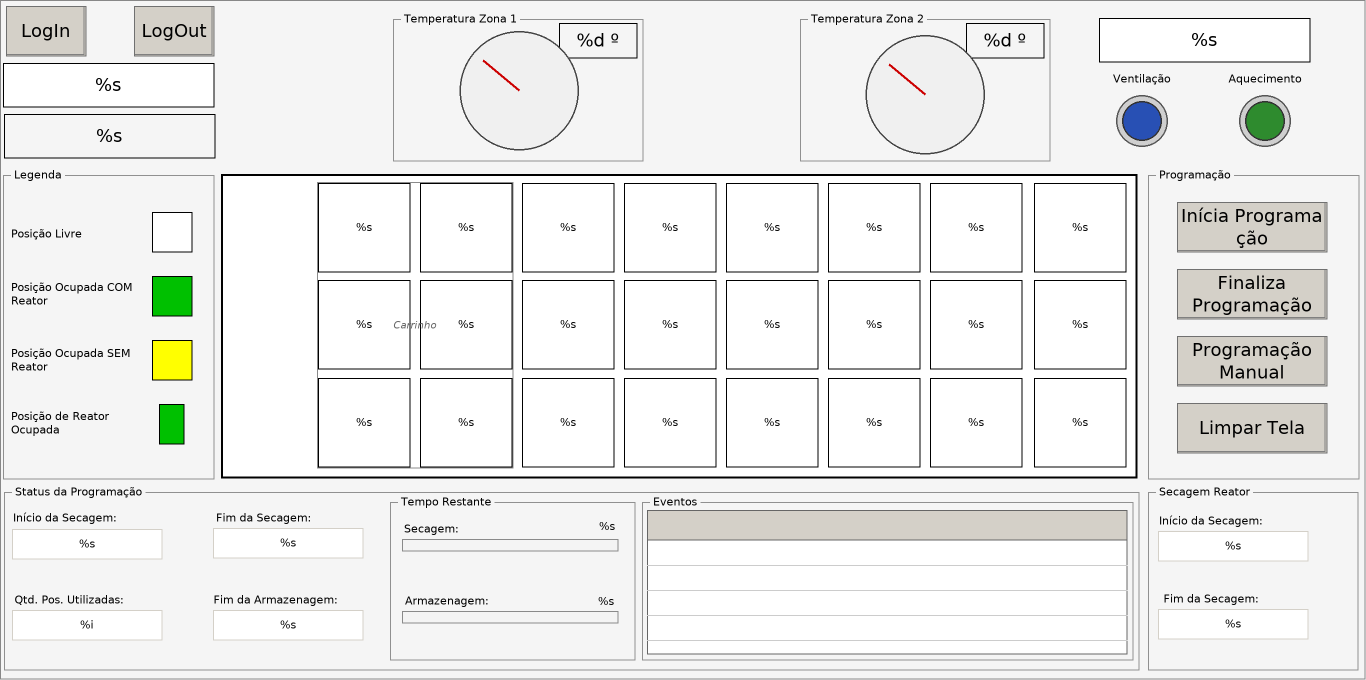
VISUALIZATION Estufa1  // 1366x680
    GroupBox (1148,484 210x186), "Secagem Reator", invisible if: GVL_P.bCarrinhoReator1
        Label (10,100 106x30), "Fim da Secagem:"
        Textfield (10,125 150x30), "%s", text variable: GVL_P.arrStatusEstufas[0].statusFimSecagem
    GroupBox (3,167 211x312), "Legenda"
        RoundedRectangle (149,173 40x40)
        RoundedRectangle (149,45 40x40)
        RoundedRectangle (156,237 25x40)
    GroupBox (800,11 250x150), "Temperatura Zona 2"
        Rectangle (166,12 78x35), "%d º", text variable: GVL.zona2atual_019
    GroupBox (393,11 250x150), "Temperatura Zona 1"
        Rectangle (166,12 78x35), "%d º", text variable: GVL.zona1atual_019
    GroupBox (4,484 1135x186), "Status da Programação"
        Label (209,19 101x30), "Fim da Secagem:"
        Label (209,101 125x30), "Fim da Armazenagem:"
        Label (8,101 114x30), "Qtd. Pos. Utilizadas:"
        GroupBox (638,10 491x166), "Eventos"
            Table (5,16 480x144), data array: GVL_P.arrLogEstufa19
                p3854506369: GVL_P.arrLogEstufa19[INDEX]
            InvisibleInput (6,17 431x142)
                OnMouseClick: OpenDialog Dialog=addComment, OpenModal=True, OpenCentered=True
        Label (8,19 106x30), "Início da Secagem:"
        Textfield (8,126 150x30), "%i", text variable: GVL.totalPos[0]
        Textfield (209,44 150x30), "%s", text variable: GVL_P.arrStatusEstufas[0].statusFimSecagem
        Textfield (209,126 150x30), "%s", text variable: GVL_P.arrStatusEstufas[0].statusFimArmazenagem
        GroupBox (386,10 245x166), "Tempo Restante"
            Progressbar (12,117 216x12), variable: MAIN.bardintArm19
            Rectangle (131,99 96x17), "%s", text variable: mid(str:=time_to_string(GVL.endArm19), LEN:= 20, POS:= 3)
            Progressbar (12,45 216x12), variable: MAIN.bardintSec19
        Label (398,30 59x30), "Secagem:"
    Rectangle (221,174 916x304)
    Rectangle (1034,183 92x89), "%s", text variable: GVL_P.aPositionsE019[1].text, colour variable: GVL_P.aPositionsE019[1].color
        OnMouseUp: OpenDialog Dialog=ConfigPosicao, Parameters={bReator: , iOFnumber: , iSrlNumber: }, OpenModal=True, OpenCentered=True
        OnMouseUp: execute {
            gvl.actPos:= 1;
            //selectPos019();
        }
    Rectangle (1034,280 92x89), "%s", text variable: GVL_P.aPositionsE019[2].text, colour variable: GVL_P.aPositionsE019[2].color
        OnMouseUp: OpenDialog Dialog=ConfigPosicao, Parameters={bReator: , iOFnumber: , iSrlNumber: }, OpenModal=True, OpenCentered=True
        OnMouseUp: execute {
            gvl.actPos:= 2;
            //selectPos019();
        }
    Rectangle (1034,378 92x89), "%s", text variable: GVL_P.aPositionsE019[3].text, colour variable: GVL_P.aPositionsE019[3].color
        OnMouseUp: OpenDialog Dialog=ConfigPosicao, Parameters={bReator: , iOFnumber: , iSrlNumber: }, OpenModal=True, OpenCentered=True
        OnMouseUp: execute {
            gvl.actPos:= 3;
            //selectPos019();
        }
    Rectangle (930,183 92x89), "%s", text variable: GVL_P.aPositionsE019[4].text, colour variable: GVL_P.aPositionsE019[4].color
        OnMouseUp: OpenDialog Dialog=ConfigPosicao, Parameters={bReator: , iOFnumber: , iSrlNumber: }, OpenModal=True, OpenCentered=True
        OnMouseUp: execute {
            gvl.actPos:= 4;
            //selectPos019();
        }
    Rectangle (930,280 92x89), "%s", text variable: GVL_P.aPositionsE019[5].text, colour variable: GVL_P.aPositionsE019[5].color
        OnMouseUp: OpenDialog Dialog=ConfigPosicao, Parameters={bReator: , iOFnumber: , iSrlNumber: }, OpenModal=True, OpenCentered=True
        OnMouseUp: execute {
            gvl.actPos:= 5;
            //selectPos019();
        }
    Rectangle (930,378 92x89), "%s", text variable: GVL_P.aPositionsE019[6].text, colour variable: GVL_P.aPositionsE019[6].color
        OnMouseUp: OpenDialog Dialog=ConfigPosicao, Parameters={bReator: , iOFnumber: , iSrlNumber: }, OpenModal=True, OpenCentered=True
        OnMouseUp: execute {
            gvl.actPos:= 6;
            //selectPos019();
        }
    Rectangle (828,183 92x89), "%s", text variable: GVL_P.aPositionsE019[7].text, colour variable: GVL_P.aPositionsE019[7].color
        OnMouseUp: OpenDialog Dialog=ConfigPosicao, Parameters={bReator: , iOFnumber: , iSrlNumber: }, OpenModal=True, OpenCentered=True
        OnMouseUp: execute {
            gvl.actPos:= 7;
            //selectPos019();
        }
    Rectangle (828,280 92x89), "%s", text variable: GVL_P.aPositionsE019[8].text, colour variable: GVL_P.aPositionsE019[8].color
        OnMouseUp: OpenDialog Dialog=ConfigPosicao, Parameters={bReator: , iOFnumber: , iSrlNumber: }, OpenModal=True, OpenCentered=True
        OnMouseUp: execute {
            gvl.actPos:= 8;
            //selectPos019();
        }
    Rectangle (828,378 92x89), "%s", text variable: GVL_P.aPositionsE019[9].text, colour variable: GVL_P.aPositionsE019[9].color
        OnMouseUp: OpenDialog Dialog=ConfigPosicao, Parameters={bReator: , iOFnumber: , iSrlNumber: }, OpenModal=True, OpenCentered=True
        OnMouseUp: execute {
            gvl.actPos:= 9;
            //selectPos019();
        }
    Rectangle (726,183 92x89), "%s", text variable: GVL_P.aPositionsE019[10].text, colour variable: GVL_P.aPositionsE019[10].color
        OnMouseUp: OpenDialog Dialog=ConfigPosicao, Parameters={bReator: , iOFnumber: , iSrlNumber: }, OpenModal=True, OpenCentered=True
        OnMouseUp: execute {
            gvl.actPos:= 10;
            //selectPos019();
        }
    Rectangle (726,280 92x89), "%s", text variable: GVL_P.aPositionsE019[11].text, colour variable: GVL_P.aPositionsE019[11].color
        OnMouseUp: OpenDialog Dialog=ConfigPosicao, Parameters={bReator: , iOFnumber: , iSrlNumber: }, OpenModal=True, OpenCentered=True
        OnMouseUp: execute {
            gvl.actPos:= 11;
            //selectPos019();
        }
    Rectangle (726,378 92x89), "%s", text variable: GVL_P.aPositionsE019[12].text, colour variable: GVL_P.aPositionsE019[12].color
        OnMouseUp: OpenDialog Dialog=ConfigPosicao, Parameters={bReator: , iOFnumber: , iSrlNumber: }, OpenModal=True, OpenCentered=True
        OnMouseUp: execute {
            gvl.actPos:= 12;
            //selectPos019();
        }
    Rectangle (624,183 92x89), "%s", text variable: GVL_P.aPositionsE019[13].text, colour variable: GVL_P.aPositionsE019[13].color
        OnMouseUp: OpenDialog Dialog=ConfigPosicao, Parameters={bReator: , iOFnumber: , iSrlNumber: }, OpenModal=True, OpenCentered=True
        OnMouseUp: execute {
            gvl.actPos:= 13;
            //selectPos019();
        }
    Rectangle (624,280 92x89), "%s", text variable: GVL_P.aPositionsE019[14].text, colour variable: GVL_P.aPositionsE019[14].color
        OnMouseUp: OpenDialog Dialog=ConfigPosicao, Parameters={bReator: , iOFnumber: , iSrlNumber: }, OpenModal=True, OpenCentered=True
        OnMouseUp: execute {
            gvl.actPos:= 14;
            //selectPos019();
        }
    Rectangle (624,378 92x89), "%s", text variable: GVL_P.aPositionsE019[15].text, colour variable: GVL_P.aPositionsE019[15].color
        OnMouseUp: OpenDialog Dialog=ConfigPosicao, Parameters={bReator: , iOFnumber: , iSrlNumber: }, OpenModal=True, OpenCentered=True
        OnMouseUp: execute {
            gvl.actPos:= 15;
            //selectPos019();
        }
    Rectangle (522,183 92x89), "%s", text variable: GVL_P.aPositionsE019[16].text, colour variable: GVL_P.aPositionsE019[16].color
        OnMouseUp: OpenDialog Dialog=ConfigPosicao, Parameters={bReator: , iOFnumber: , iSrlNumber: }, OpenModal=True, OpenCentered=True
        OnMouseUp: execute {
            gvl.actPos:= 16;
            //selectPos019();
        }
    Rectangle (522,280 92x89), "%s", text variable: GVL_P.aPositionsE019[17].text, colour variable: GVL_P.aPositionsE019[17].color
        OnMouseUp: OpenDialog Dialog=ConfigPosicao, Parameters={bReator: , iOFnumber: , iSrlNumber: }, OpenModal=True, OpenCentered=True
        OnMouseUp: execute {
            gvl.actPos:= 17;
            //selectPos019();
        }
    Rectangle (522,378 92x89), "%s", text variable: GVL_P.aPositionsE019[18].text, colour variable: GVL_P.aPositionsE019[18].color
        OnMouseUp: OpenDialog Dialog=ConfigPosicao, Parameters={bReator: , iOFnumber: , iSrlNumber: }, OpenModal=True, OpenCentered=True
        OnMouseUp: execute {
            gvl.actPos:= 18;
            //selectPos019();
        }
    Rectangle (420,183 92x89), "%s", text variable: GVL_P.aPositionsE019[19].text, colour variable: GVL_P.aPositionsE019[19].color
        OnMouseUp: OpenDialog Dialog=ConfigPosicao, Parameters={bReator: , iOFnumber: , iSrlNumber: }, OpenModal=True, OpenCentered=True
        OnMouseUp: execute {
            gvl.actPos:= 19;
            //selectPos019();
        }
    Rectangle (420,280 92x89), "%s", text variable: GVL_P.aPositionsE019[20].text, colour variable: GVL_P.aPositionsE019[20].color
        OnMouseUp: OpenDialog Dialog=ConfigPosicao, Parameters={bReator: , iOFnumber: , iSrlNumber: }, OpenModal=True, OpenCentered=True
        OnMouseUp: execute {
            gvl.actPos:= 20;
            //selectPos019();
        }
    Rectangle (420,378 92x89), "%s", text variable: GVL_P.aPositionsE019[21].text, colour variable: GVL_P.aPositionsE019[21].color
        OnMouseUp: OpenDialog Dialog=ConfigPosicao, Parameters={bReator: , iOFnumber: , iSrlNumber: }, OpenModal=True, OpenCentered=True
        OnMouseUp: execute {
            gvl.actPos:= 21;
            //selectPos019();
        }
    Rectangle (318,183 92x89), "%s", text variable: GVL_P.aPositionsE019[22].text, colour variable: GVL_P.aPositionsE019[22].color
        OnMouseUp: OpenDialog Dialog=ConfigPosicao, Parameters={bReator: , iOFnumber: , iSrlNumber: }, OpenModal=True, OpenCentered=True
        OnMouseUp: execute {
            gvl.actPos:= 22;
            //selectPos019();
        }
    Rectangle (318,280 92x89), "%s", text variable: GVL_P.aPositionsE019[23].text, colour variable: GVL_P.aPositionsE019[23].color
        OnMouseUp: OpenDialog Dialog=ConfigPosicao, Parameters={bReator: , iOFnumber: , iSrlNumber: }, OpenModal=True, OpenCentered=True
        OnMouseUp: execute {
            gvl.actPos:= 23;
            //selectPos019();
        }
    Rectangle (318,378 92x89), "%s", text variable: GVL_P.aPositionsE019[24].text, colour variable: GVL_P.aPositionsE019[24].color
        OnMouseUp: OpenDialog Dialog=ConfigPosicao, Parameters={bReator: , iOFnumber: , iSrlNumber: }, OpenModal=True, OpenCentered=True
        OnMouseUp: execute {
            gvl.actPos:= 24;
            //selectPos019();
        }
    Meter180 (399,31 240x119), value: GVL.zona1atual_019, style: Meter-Meter180-Gray, scale format: %.1f, scale 20..160
        p518627256: ºC
    GroupBox (1148,167 211x312), "Programação"
        Button (29,35 150x50), "Inícia Programação", input disabled if: GVL_P.arrStatusEstufas[GVL.actEst].start
            OnMouseClick: OpenDialog Dialog=IniciaProg, OpenModal=True, OpenCentered=True
            OnMouseClick: execute { iniciaProgramacaoEstufa(); }
        Button (29,102 150x50), "Finaliza Programação"
            OnMouseClick: OpenDialog Dialog=FinalizaProg, Parameters={bReator: , iOFnumber: , iSrlNumber: }, OpenModal=True, OpenCentered=True
        Button (29,169 150x50), "Programação Manual", input disabled if: GVL_P.arrStatusEstufas[GVL.actEst].start
            OnMouseClick: OpenDialog Dialog=TimeCustom, OpenModal=True, OpenCentered=True
            OnMouseClick: execute { iniciaProgramacaoEstufa(); }
    Textfield (12,529 150x30), "%s", text variable: GVL_P.arrStatusEstufas[0].statusInicioSecagem
    Label (402,586 90x30), "Armazenagem:"
    Meter180 (805,35 240x119), value: GVL.zona2atual_019, style: Meter-Meter180-Gray, scale format: %.1f, scale 20..160
        p518627256: ºC
    RoundedRectangle (152,276 40x40)
    Label (8,278 132x32), "Posição Ocupada COM Reator"
    Label (8,344 128x32), "Posição Ocupada SEM Reator"
    Label (8,218 84x32), "Posição Livre"
    Label (8,407 128x32), "Posição de Reator Ocupada"
    Frame (317,182 196x286), invisible if: GVL_P.bCarrinhoReator1
        shows Carrinho()
    Rectangle (3,63 211x44), "%s", text variable: MAIN.sDB_Operador
    Lamp1 (1112,91 60x60), variable: GVL.ventilacao_Ligada_019, style: Lamp-Lamp1-Blue
    Lamp1 (1235,91 60x60), variable: GVL.aquecimento_Ligado_019, style: Lamp-Lamp1-Green
    Label (1108,64 68x30), "Ventilação"
    Label (1227,64 76x30), "Aquecimento"
    Textfield (1158,531 150x30), "%s", text variable: GVL_P.arrStatusEstufas[0].inicioReator, invisible if: GVL_P.bCarrinhoReator1
    Label (1158,506 106x30), "Início da Secagem:", invisible if: GVL_p.bCarrinhoReator1
    Rectangle (1099,18 211x44), "%s", text variable: GVL_P.etapa_process[GVL.actEst]
    Rectangle (522,518 96x17), "%s", text variable: mid(str:=time_to_string(GVL.endSeca19), LEN:= 20, POS:= 3)
    Rectangle (4,114 211x44), "%s", text variable: GVL.sSystemTime
    Button (1177,403 150x50), "Limpar Tela"
        OnMouseClick: execute {
            FOR gvl.i:=1 TO 24 BY 1 DO
            gvl_p.aPositionsE019[gvl.i].numOF:='';
            gvl_p.aPositionsE019[gvl.i].lote:='';
            gvl_p.aPositionsE019[gvl.i].class:=0;
            gvl_p.aPositionsE019[gvl.i].pot:=0;
            gvl_p.aPositionsE019[gvl.i].cor:=0;
            gvl_p.aPositionsE019[gvl.i].text:='';
            gvl_p.aPositionsE019[gvl.i].reator:=true;
            END_FOR
            FOR gvl.i:=1 TO 18 BY 1 DO
            gvl_p.corPosReator1[gvl.i].cor:=0;
            END_FOR
            gravarConfigPosicao.bReator[0]:= false;
            ///// GERADOR DE LOG -------------------------------------------------------------
            gvl.envialog:= 'Todas as posições foram limpas. ESTUFA 19';
            gvl.logRegister19:= gvl.envialog;
            gvl.sCmdInsertLog:= 'INSERT INTO [dbo].[LogGeneral] ([HistoricalTime],[Description])VALUES($'$',$'$')';
            gvl.sCmdInsertLog:= insert(gvl.sCmdInsertLog,gvl.logRegister19,74);
            gvl.sCmdInsertLog:= insert(gvl.sCmdInsertLog,gvl.sSystemDateTime,71);
            gvl.bInsertLog:= TRUE;
        }
    Button (6,6 80x50), "LogIn"
        OnMouseClick: VisuUserMgmt Type=Login
        OnMouseClick: execute { gvl.logButton:= true; }
    Button (134,6 80x50), "LogOut"
        OnMouseClick: VisuUserMgmt Type=Logout
        OnMouseClick: execute { gvl.logButton:= false; }
END_VISUALIZATION

(* stored: Version 1.1.0.1, ProductVersion 3.1.4024.12
   Visu Estufa1: Id {4ca0d67f-7005-4db2-a762-a1c17892b4ec} *)
